Universal Robots PolyScope program: Test Teach Sleeve Fillet.urp

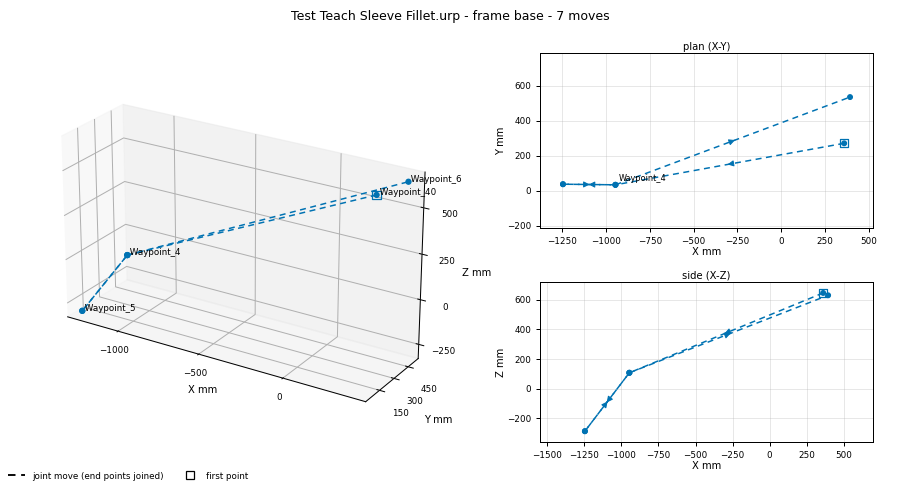
[picture p0: tool path of Test Teach Sleeve Fillet.urp in frame base, 7 of 7 moves have a stored position in this frame; points joined in program order, loops and branches not executed]
Program Test Teach Sleeve Fillet (installation=default directory=/programs createdIn=5.21.3 lastSavedIn=5.21.3 robotSerialNumber=20246801938)
Calibrated DH parameters: a=[-0.000071, -0.790281, -0.600694, 0.000061, -0.000039, 0]; d=[0.236272, 604.465945, 132.116513, -736.382239, 0.159268, 0.154005]; alpha=[1.570254, -0.000567, 0.000559, 1.571709, -1.56999, 0]; deltaTheta=[0, -0.409357, 7.293326, -0.600784, -0.000001, -0.000001]
InitVariablesNode variables(variable(name=free_dr_already, expression=False), variable(name=freedrive_m_var, expression=False))
Robot Program (runOnlyOnce=false)
  Set NoAction tcp=pretend_w_top
  SuppressedNode
    MoveL speed 250 mm/s, acceleration 1200 mm/s^2 (useActiveTCP=true optimoveEnabled=false optiMoveSpeed=0.3 optiMoveAcceleration=0.09) feature=Base
      Waypoint Waypoint_1: TCP in base x=183.613 y=373.491 z=464.002 mm, rx=0 ry=3.1416 rz=0 rad; joints [-144.817, -120.486, 148.461, -117.931, -90.033, 125.101] deg; TCP offset x=0 y=0 z=19 mm, rx=0 ry=0 rz=0 rad
      'move welder up out of holder'
  MoveJ speed 60 deg/s, acceleration 80 deg/s^2 (useActiveTCP=false optimoveEnabled=false optiMoveSpeed=0.3 optiMoveAcceleration=0.09) tcp=TCP_1_plate; feature=Base
    Waypoint Waypoint_40: TCP in base x=360.688 y=270.12 z=646.145 mm, rx=0.0578 ry=2.126 rz=2.1341 rad; joints [-198.126, -117.852, 133.303, -13.01, -11.422, -6.036] deg
    'above waypoint is home'
    SuppressedNode
      Waypoint Waypoint_2: TCP in base x=-548.957 y=386.285 z=143.71 mm, rx=1.5708 ry=0 rz=0 rad; joints [-60.253, -57.926, 123.544, -65.529, -60.311, -0.099] deg
    SuppressedNode
      Waypoint Waypoint_3: TCP in base x=-565.561 y=-88.282 z=748.934 mm, rx=0.347 ry=3.1015 rz=-0.0385 rad; joints [-12.028, -113.359, 121.362, 263.351, -88.693, -89.284] deg
    Waypoint Waypoint_4: TCP in base x=-946.63 y=32.923 z=107.553 mm, rx=1.1855 ry=-1.4546 rz=-1.2991 rad; joints [-14.723, -32.384, 121.91, 97.274, -87.344, -180.783] deg
  Set NoAction tcp=pretend_w_top
  freedrive_m_var := False
  freedrive_m_var := True
  Popup Message (haltProgram=false message=Move the TCP to point 1 on the edge then click 'Continue' inputType=Text)
  tcp_pose_left := get_actual_tcp_pose()
  freedrive_m_var := False
  Script: sync()
  Wait Sleep waitTime=0.01
  MoveJ speed 60 deg/s, acceleration 80 deg/s^2 (useActiveTCP=true optimoveEnabled=false optiMoveSpeed=0.3 optiMoveAcceleration=0.09) feature=Base
    Waypoint Waypoint_4: TCP in base x=-946.63 y=32.923 z=107.553 mm, rx=1.1855 ry=-1.4546 rz=-1.2991 rad; joints [-14.723, -32.384, 121.91, 97.274, -87.344, -180.783] deg
  MoveJ speed 60 deg/s, acceleration 80 deg/s^2 (useActiveTCP=true optimoveEnabled=false optiMoveSpeed=0.3 optiMoveAcceleration=0.09) feature=Base
    Waypoint Waypoint_5: TCP in base x=-1246.557 y=36.36 z=-286.524 mm, rx=0.3629 ry=-1.2595 rz=-1.7222 rad; joints [1.222, -11.211, 100.501, 238.355, -233.303, -3.079] deg; TCP offset x=-1.032 y=-18.062 z=285.234 mm, rx=0 ry=0 rz=0 rad
  freedrive_m_var := True
  Popup Message (haltProgram=false message=Move the TCP to point 2 on the edge then click 'Continue' inputType=Text)
  tcp_pose_right := get_actual_tcp_pose()
  Popup Message (haltProgram=false message=Move the TCP to point 3 on the edge then click 'Continue' inputType=Text)
  tcp_3 := get_actual_tcp_pose()
  freedrive_m_var := False
  Wait Sleep waitTime=0.25
  Script: sync()
  MoveL speed 100 mm/s, acceleration 1200 mm/s^2 (useActiveTCP=true optimoveEnabled=false optiMoveSpeed=0.3 optiMoveAcceleration=0.09) feature=Base
    MoveDirectionNode expression=[1.0,0.0,-0.5]
      Until DISTANCE (allowActions=false deceleration=3 distanceNodeType=STOP) Distance=0.15; motionParameters(blendRadius=0)
  MoveJ speed 60 deg/s, acceleration 80 deg/s^2 (useActiveTCP=true optimoveEnabled=false optiMoveSpeed=0.3 optiMoveAcceleration=0.09) feature=Base
    Waypoint Waypoint_5: TCP in base x=-1246.557 y=36.36 z=-286.524 mm, rx=0.3629 ry=-1.2595 rz=-1.7222 rad; joints [1.222, -11.211, 100.501, 238.355, -233.303, -3.079] deg
    Waypoint Waypoint_4: TCP in base x=-946.63 y=32.923 z=107.553 mm, rx=1.1855 ry=-1.4546 rz=-1.2991 rad; joints [-14.723, -32.384, 121.91, 97.274, -87.344, -180.783] deg; TCP offset x=0 y=0 z=19 mm, rx=0 ry=0 rz=0 rad
    Waypoint Waypoint_6: TCP in base x=394.188 y=534.376 z=630.191 mm, rx=0.0578 ry=2.126 rz=2.1341 rad; joints [-198.279, -117.801, 133.277, -12.745, -11.485, -6.332] deg; TCP offset x=-1.032 y=-18.062 z=285.234 mm, rx=0 ry=0 rz=0 rad
Thread Thread_1 (runOnlyOnce=true)
  Loop While (checkContinuously=false) expression=True
    If freedrive_m_var≟ True
      Script: freedrive_mode()
      free_dr_already := True
    Else 
      If free_dr_already
        Script: end_freedrive_mode()
        free_dr_already := False
    Script: sync()
